(* PLC project Basic_Com, Beckhoff Automation GmbH TwinCAT PLC Control 3.5.13.20 *)
(* stored: creationDateTime 2026-02-18T19:23:56.308572, modificationDateTime 2026-02-18T19:23:56.308572 *)

FUNCTION_BLOCK ProgramMain
  VAR_INPUT
    ESTOP : BOOL := FALSE;
    START : BOOL := FALSE;
    STOP : BOOL := FALSE;
  END_VAR
  VAR_OUTPUT
    MOTOR : BOOL := FALSE;
  END_VAR
  VAR_IN_OUT
    RUN : BOOL := FALSE;
  END_VAR

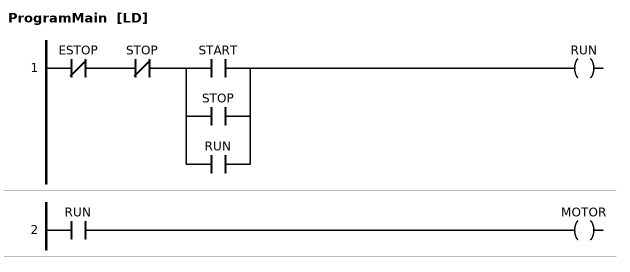
(* LD diagram, written out as Structured Text *)
RUN := NOT ESTOP AND NOT STOP AND (START OR STOP OR RUN);
MOTOR := RUN;
END_FUNCTION_BLOCK
